FUNCTION_BLOCK fbBasicRunnerTests
VAR
	runs : UINT;	
END_VAR

{attribute 'TcRpcEnable'}
METHOD ResetCounter : UINT
runs := 0;
END_METHOD

{attribute 'TcRpcEnable'}
METHOD RunCount : UINT
runs := runs + 1;
RunCount := runs;
END_METHOD

{attribute 'TcRpcEnable'}
METHOD RunUntilReturnsTrue : BOOL
VAR_INPUT
	_m : BOOL;
END_VAR
RunUntilReturnsTrue := _m;
END_METHOD

END_FUNCTION_BLOCK

(* stored: Version 1.1.0.1, ProductVersion 3.1.4024.4
   POU fbBasicRunnerTests: Id {fd9c95ca-8e53-463c-8da7-85668c18933c}, SpecialFunc None
   Method ResetCounter: Id {69f038ce-3e8e-44f5-ab3f-68781d9515df}
   Method RunCount: Id {86e50e4e-25cb-4738-89df-2c471d24676b}
   Method RunUntilReturnsTrue: Id {b9fe7b38-c5bd-482a-987b-e6f26e72a83b} *)
